FUNCTION_BLOCK POU
VAR_INPUT
END_VAR
VAR_OUTPUT
END_VAR
VAR
END_VAR

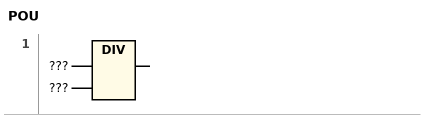
// NETWORK 1
(* ??? / ???; result not used *)

END_FUNCTION_BLOCK

(* stored: Version 1.1.0.1, ProductVersion 3.1.4024.15
   POU POU: Id {5df4d096-1806-42cb-a58c-dd6d4cfd498f}, SpecialFunc None *)
